FUNCTION_BLOCK SPLIT_AW_INTO_AB (* this Function splits the 2 AB (BYTE) adapters from a AW (WORD) *)
  (* Standard: 61499-2; Description: Copyright (c) 2026 Meisterschulen am Ostbahnhof SPDX-License-Identifier: EPL-2.0 *)
  (* Version 1.0, 2026-05-16, Franz Höpfinger, Meisterschulen am Ostbahnhof, initial API and implementation and/or initial documentation *)
  PACKAGE adapter::splitting;
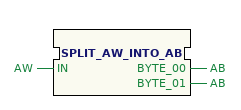
  SOCKETS
    IN : adapter::types::unidirectional::AW; (* WORD Input *)
  END_SOCKETS
  PLUGS
    BYTE_00 : adapter::types::unidirectional::AB; (* Byte 0 *)
    BYTE_01 : adapter::types::unidirectional::AB; (* Byte 1 *)
  END_PLUGS
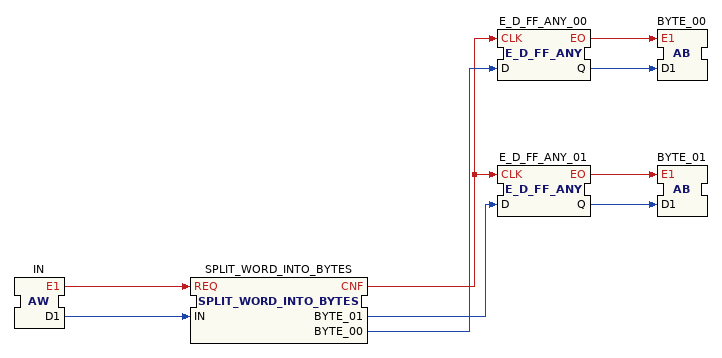
  FBS
    E_D_FF_ANY_00 : iec61499::events::E_D_FF_ANY;
    E_D_FF_ANY_01 : iec61499::events::E_D_FF_ANY;
    SPLIT_WORD_INTO_BYTES : eclipse4diac::utils::splitting::SPLIT_WORD_INTO_BYTES;
  END_FBS
  EVENT_CONNECTIONS
    IN.E1 TO SPLIT_WORD_INTO_BYTES.REQ;
    SPLIT_WORD_INTO_BYTES.CNF TO E_D_FF_ANY_00.CLK;
    SPLIT_WORD_INTO_BYTES.CNF TO E_D_FF_ANY_01.CLK;
    E_D_FF_ANY_00.EO TO BYTE_00.E1;
    E_D_FF_ANY_01.EO TO BYTE_01.E1;
  END_CONNECTIONS
  DATA_CONNECTIONS
    IN.D1 TO SPLIT_WORD_INTO_BYTES.IN;
    SPLIT_WORD_INTO_BYTES.BYTE_01 TO E_D_FF_ANY_01.D;
    SPLIT_WORD_INTO_BYTES.BYTE_00 TO E_D_FF_ANY_00.D;
    E_D_FF_ANY_00.Q TO BYTE_00.D1;
    E_D_FF_ANY_01.Q TO BYTE_01.D1;
  END_CONNECTIONS
END_FUNCTION_BLOCK
